FUNCTION_BLOCK Port (* Service Interface Function Block Type *)
  (* Standard: 61499-2; Description: Copyright (c) 2021 Jonathan Lainer This program and the accompanying materials are made available under the terms of the Eclipse Public License 2.0 which is available at https://www.eclipse.org/legal/epl-2.0/ SPDX-License-Identifier: EPL-2.0 *)
  (* Version 1.0, 2021-02-22, Jonathan Lainer, Initial Contribution *)
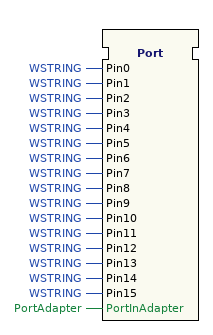
  VAR_INPUT
    Pin0 : WSTRING; (* Name of the Pin *)
    Pin1 : WSTRING; (* Name of the Pin *)
    Pin2 : WSTRING; (* Name of the Pin *)
    Pin3 : WSTRING; (* Name of the Pin *)
    Pin4 : WSTRING; (* Name of the Pin *)
    Pin5 : WSTRING; (* Name of the Pin *)
    Pin6 : WSTRING; (* Name of the Pin *)
    Pin7 : WSTRING; (* Name of the Pin *)
    Pin8 : WSTRING; (* Name of the Pin *)
    Pin9 : WSTRING; (* Name of the Pin *)
    Pin10 : WSTRING; (* Name of the Pin *)
    Pin11 : WSTRING; (* Name of the Pin *)
    Pin12 : WSTRING; (* Name of the Pin *)
    Pin13 : WSTRING; (* Name of the Pin *)
    Pin14 : WSTRING; (* Name of the Pin *)
    Pin15 : WSTRING; (* Name of the Pin *)
  END_VAR
  SOCKETS
    PortInAdapter : PortAdapter;
  END_SOCKETS
END_FUNCTION_BLOCK
